(* IEC 61131-3 sources: statemachine/src/StateFramework/Transitions, 2 files *)

(* ---- ITransition.st ---- *)
NAMESPACE Simatic.Ax.StateFramework
    INTERFACE ITransition

        // Returns the guard that decides whether the transition may fire.
        METHOD GetGuard : IGuard
        END_METHOD

        // Returns the target state that becomes active after the transition.
        METHOD GetNextState : IState
        END_METHOD

    END_INTERFACE

    INTERFACE IMutableTransition

        // Configures guard and target state in one call.
        METHOD Config
            VAR_INPUT
                g : IGuard;
                ns : IState;
            END_VAR
        END_METHOD

    END_INTERFACE
END_NAMESPACE

(* ---- Transition.st ---- *)
NAMESPACE Simatic.Ax.StateFramework
    CLASS Transition IMPLEMENTS ITransition, IMutableTransition

        VAR PUBLIC
            Guard : IGuard;
            NextState : IState;
        END_VAR

        METHOD PUBLIC GetGuard : IGuard
            GetGuard := Guard;
        END_METHOD

        METHOD PUBLIC GetNextState : IState
            GetNextState := NextState;
        END_METHOD

        METHOD PUBLIC Config
            VAR_INPUT
                g : IGuard;
                ns : IState;
            END_VAR
            // Config wires a guard and its target state in one call.
            Guard := g;
            NextState := ns;
        END_METHOD

    END_CLASS
END_NAMESPACE
